PROGRAM MAIN
VAR
	bStart : BOOL := FALSE;
    bStop : BOOL := FALSE;
    bAlarm : BOOL := FALSE;
    iCounter : INT := 0;
    rTemperature : REAL := 30.0;
END_VAR


IF bStart THEN
    iCounter := iCounter + 1;
    rTemperature := rTemperature + 0.1;
END_IF

IF rTemperature > 40.0 THEN
    bAlarm := TRUE;
END_IF

IF bStop THEN
    bStart := FALSE;
    rTemperature := 30.0;
    bAlarm := FALSE;
    iCounter := 0;
END_IF

END_PROGRAM

(* stored: Version 1.1.0.1, ProductVersion 3.1.4024.15
   POU MAIN: Id {c61b1abb-271f-4af8-bb84-09a656ce1d2d}, SpecialFunc None *)
